// TIA Portal project "P2" (V15.1)

(* hardware
DEVICE "ET 200SP station_2"  ET 200SP-Station
   slot 0: "Rack_0"  Rack  6ES5 710-8MAx1
   slot 1: "PLC_1"  CPU 1512SP F-1 PN  6ES7 512-1SK01-0AB0  V2.6
   slot 2: "DI 8x24VDC HF_1"  DI 8x24VDC HF  6ES7 131-6BF00-0CA0  V2.0
      slot 1: "DI 8x24VDC HF_1"  DI 8x24VDC HF
   slot 3: "DI 8x24VDC HF_2"  DI 8x24VDC HF  6ES7 131-6BF00-0CA0  V2.0
      slot 1: "DI 8x24VDC HF_2"  DI 8x24VDC HF
   slot 4: "DQ 8x24VDC/0.5A HF_1"  DQ 8x24VDC/0.5A HF  6ES7 132-6BF00-0CA0  V2.0
      slot 1: "DQ 8x24VDC/0.5A HF_1"  DQ 8x24VDC/0.5A HF
   slot 5: "DQ 8x24VDC/0.5A HF_2"  DQ 8x24VDC/0.5A HF  6ES7 132-6BF00-0CA0  V2.0
      slot 1: "DQ 8x24VDC/0.5A HF_2"  DQ 8x24VDC/0.5A HF
   slot 6: "CM 4xIO-Link_1"  CM 4xIO-Link  6ES7 137-6BD00-0BA0  V2.2
      slot 1: "CM 4xIO-Link_1"  6ES7 137-6BD00-0BA0
   slot 7: "Server module_1"  Server module  6ES7 193-6PA00-0AA0  V1.1
      slot 1: "Server module_1"  Server module
   slot 127: "BA 2xRJ45"  BA 2xRJ45  6ES7 193-6AR00-0AA0  V0.0
      slot 32769: "Port_1"  6ES7 193-6AR00-0AA0
      slot 32770: "Port_2"  6ES7 193-6AR00-0AA0
*)

// ===== PLC "PLC_1"  CPU 1512SP F-1 PN =====

VAR_GLOBAL   // PLC tag table "gtConv_tag table"
   "start_btn" AT %I1.0 : Bool;
   "stop_btn" AT %I1.1 : Bool;
   "select_op_mode" AT %I1.2 : Bool;
   "reset_btn" AT %I1.3 : Bool;
   "carr_det_stop_pos" AT %I1.4 : Bool;
   "EM_stop" AT %I1.5 : Bool;
   "carr_det_conv_entry" AT %I1.6 : Bool;
   "carr_det_conv_exit" AT %I1.7 : Bool;
   "Carr_id_bit0_det" AT %I42.0 : Bool;
   "Carr_id_bit1_det" AT %I42.1 : Bool;
   "Carr_id_bit2_det" AT %I42.2 : Bool;
   "Carr_id_bit3_det" AT %I42.3 : Bool;
   "SW_s1" AT %I42.4 : Bool;
   "SW_s2" AT %I42.5 : Bool;
   "stop_cyl_low_end" AT %I42.7 : Bool;
   "SW_start_light" AT %Q1.0 : Bool;
   "SW_reset_light" AT %Q1.1 : Bool;
   "SW_func_Q1_light" AT %Q1.2 : Bool;
   "SW_func_Q2_light" AT %Q1.3 : Bool;
   "belt_forward" AT %Q1.4 : Bool;
   "belt_reverse" AT %Q1.5 : Bool;
   "select_belt_speed" AT %Q1.6 : Bool;
   "stop_cyl_mov_down" AT %Q1.7 : Bool;
   "coupling_signal_left" AT %Q42.4 : Bool;
   "coupling_signal_right" AT %Q42.5 : Bool;
   "X-axix_left_end_pos" AT %I0.0 : Bool;   // DI0.0
   "X-axis_right_pos" AT %I0.1 : Bool;   // DI0.1
   "front_cover_correct" AT %I0.2 : Bool;   // DI0.2
   "front_cover_present" AT %I0.3 : Bool;   // DI0.3
   "Z-axis_upper_pos" AT %I0.4 : Bool;   // DI0.4
   "Z_axis_lower_pos" AT %I0.5 : Bool;   // DI0.5
   "back_cover_present" AT %I0.7 : Bool;   // DI0.7
   "move_X-axis_left" AT %Q0.0 : Bool;   // DQ0.0
   "move_X-axis_right" AT %Q0.1 : Bool;   // DQ0.1
   "switch_drill_1" AT %Q0.2 : Bool;   // DQ0.2
   "switch_drill_2" AT %Q0.3 : Bool;   // DQ0.3
   "move_Z-axis_up" AT %Q0.4 : Bool;   // DQ0.4
   "move_Z-axis_down" AT %Q0.5 : Bool;   // DQ0.5
   "open_Z-axis_end_pos_lock" AT %Q0.6 : Bool;   // DQ0.6
END_VAR

DATA_BLOCK "idbDriveBelt"   // DB1
{ S7_Optimized_Access := 'TRUE' }
VERSION : 0.1
// stored: InstanceOfName fbDriveBelt
"fbDriveBelt"
BEGIN
END_DATA_BLOCK

FUNCTION_BLOCK "fbDriveBelt"   // FB1, SCL
{ S7_Optimized_Access := 'TRUE' }
VERSION : 0.1
   VAR_INPUT
      bStartBtn : Bool;
      bStoppBtn : Bool;
      bConveyerEntry : Bool;
      bConveyerExit : Bool;
      bConveyerStopper : Bool;
      bResetBtn : Bool;
      "bX-axis_left" : Bool;
      "bX-axis_right" : Bool;
      "bZ-axis_up" : Bool;
      "bZ-axis_down" : Bool;
   END_VAR
   VAR
      sbStartBtnLt : Bool;
      sbBeltForward : Bool;
      sbSendForward : Bool;
      sbResetBtnLt : Bool;
      sbMoveXaxLeft : Bool;
      sbMoveXaxRight : Bool;
      sbDrill1On : Bool;
      sbDrill2On : Bool;
      sbMoveZaxUp : Bool;
      sbMoveZaxDown : Bool;
      sbOpenZaxLock : Bool;
   END_VAR
BEGIN

   IF #bStartBtn THEN
       #sbStartBtnLt := TRUE;
       #sbBeltForward := TRUE;
       #sbResetBtnLt := FALSE;
       ;
   END_IF;

   IF #bConveyerStopper THEN
       #sbMoveXaxRight := true;
       #sbMoveXaxLeft := false;
       #sbMoveZaxDown := true;
       #sbMoveZaxUp := false;
       #sbOpenZaxLock := true;
       #sbDrill1On := TRUE;
       #sbDrill2On := TRUE;
   ELSE
       #sbMoveXaxRight := FALSE;
       #sbMoveXaxLeft := TRUE;
       #sbMoveZaxDown := FALSE;
       #sbMoveZaxUp := TRUE;
       #sbDrill1On := false;
       #sbDrill2On := false;
       #sbOpenZaxLock := TRUE;
       ;
   END_IF;


   (*
   IF #bResetBtn THEN
       #sbResetBtnLt := TRUE;
       #sbBeltForward := FALSE;
       #sbStartBtnLt := FALSE;
       ;
   END_IF;
   *)

   IF #bResetBtn THEN
       #sbResetBtnLt := true;
       #sbSendForward := true;
   ELSE
       #sbResetBtnLt := false;
       #sbSendForward := false;
       ;
   END_IF;

   IF #bStoppBtn = FALSE THEN
       #sbBeltForward := FALSE;
       #sbStartBtnLt := FALSE;
       #sbResetBtnLt := FALSE;
       #sbOpenZaxLock := FALSE;
       ;
   END_IF;

   (*
   IF #bConveyerStopper THEN
       #sbSendForward := true;
       ;
   ELSE
       #sbSendForward := FALSE;
   END_IF;
   *)
   (*
   IF #bConveyerEntry THEN
       #sbBeltForward := true;
       #sbBeltReversed := false;
       ;
   END_IF;

   IF #bConveyerExit THEN
       #sbBeltReversed := TRUE;
       #sbBeltForward := FALSE;
       ;
   END_IF;
   *)
END_FUNCTION_BLOCK

ORGANIZATION_BLOCK "Main"   // OB1, SCL, ProgramCycle
TITLE = "Main Program Sweep (Cycle)"
{ S7_Optimized_Access := 'TRUE' }
VERSION : 0.1
   VAR_INPUT
      Initial_Call : Bool;   // Initial call of this OB
      Remanence : Bool;   // =True, if remanent data are available
   END_VAR
BEGIN
   //Innganger transportbånd
   "idbDriveBelt".bStartBtn := "start_btn";
   "idbDriveBelt".bStoppBtn := "stop_btn";
   "idbDriveBelt".bConveyerEntry := "carr_det_conv_entry";
   "idbDriveBelt".bConveyerExit := "carr_det_conv_exit";
   "idbDriveBelt".bConveyerStopper := "carr_det_stop_pos";
   "idbDriveBelt".bResetBtn := "reset_btn";
   "idbDriveBelt".bResetBtn := "reset_btn";

   //Utganger transportbånd
   "idbDriveBelt".sbBeltForward := "belt_forward";
   "idbDriveBelt".sbStartBtnLt := "SW_start_light";
   "idbDriveBelt".sbSendForward := "stop_cyl_mov_down";
   "idbDriveBelt".sbResetBtnLt := "SW_reset_light";
   "idbDriveBelt".sbBeltForward := "belt_forward";
   "idbDriveBelt".sbStartBtnLt := "SW_start_light";
   "idbDriveBelt".sbSendForward := "stop_cyl_mov_down";
   "idbDriveBelt".sbResetBtnLt := "SW_reset_light";

   //Innganger iDrill
   "idbDriveBelt"."bX-axis_left" := "X-axix_left_end_pos";
   "idbDriveBelt"."bX-axis_right" := "X-axis_right_pos";
   "idbDriveBelt"."bZ-axis_down" := "Z_axis_lower_pos";
   "idbDriveBelt"."bZ-axis_up" := "Z-axis_upper_pos";

   //Utganger iDrill
   "idbDriveBelt".sbMoveXaxLeft := "move_X-axis_left";
   "idbDriveBelt".sbMoveXaxRight := "move_X-axis_right";
   "idbDriveBelt".sbDrill1On := "switch_drill_1";
   "idbDriveBelt".sbDrill2On := "switch_drill_2";
   "idbDriveBelt".sbMoveZaxDown := "move_Z-axis_down";
   "idbDriveBelt".sbMoveZaxUp := "move_Z-axis_up";
   "idbDriveBelt".sbOpenZaxLock := "open_Z-axis_end_pos_lock";

   //Starter idb
   "idbDriveBelt"();

   //Utganger transportbånd
   "belt_forward" := "idbDriveBelt".sbBeltForward;
   "SW_start_light" := "idbDriveBelt".sbStartBtnLt;
   "stop_cyl_mov_down" := "idbDriveBelt".sbSendForward;
   "SW_reset_light" := "idbDriveBelt".sbResetBtnLt;

   //Utganger iDill
   "move_X-axis_left" := "idbDriveBelt".sbMoveXaxLeft;
   "move_X-axis_right" := "idbDriveBelt".sbMoveXaxRight;
   "switch_drill_1" := "idbDriveBelt".sbDrill1On;
   "switch_drill_2" := "idbDriveBelt".sbDrill2On;
   "move_Z-axis_down" := "idbDriveBelt".sbMoveZaxDown;
   "move_Z-axis_up" := "idbDriveBelt".sbMoveZaxUp;
   "open_Z-axis_end_pos_lock" := "idbDriveBelt".sbOpenZaxLock;
END_ORGANIZATION_BLOCK